RoboDK station: Artist_Larry.rdk

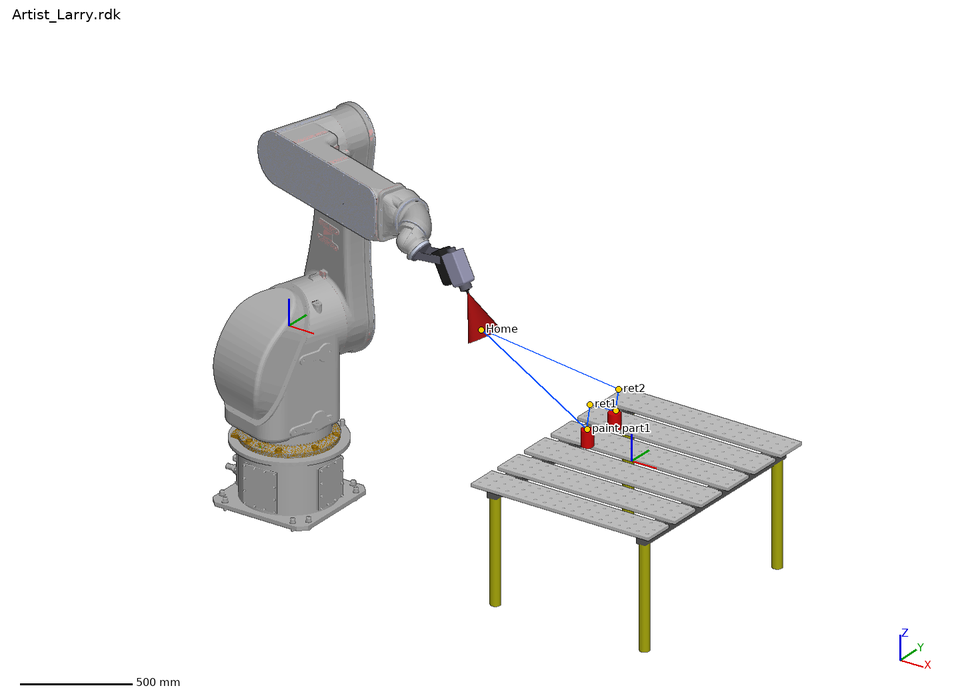
[picture v0: the station drawn from its stored meshes, robots at their saved joint values, targets as dots, program paths as lines]
Station Artist_Larry (saved by RoboDK 5.5.4). Poses are relative to the parent item; angles as X-Y-Z fixed-axis rotations.
Station parameters (name, value as stored): LIN64
  - frame Fanuc P-50iB/10L Base at (0, 0, 0) mm
    - robot Fanuc P-50iB/10L: 6 axes, payload 10 kg, reach 1800 mm, repeatability 0.2 mm, weight 331 kg
        modified DH rows (alpha deg, a mm, theta deg, d mm): 0, 0, 0, 850; -90, 0, -90, 0; 0, 900, 0, 0; -90, 0, -90, 863.603; 70, 0, 0, 106.418; -70, 0, 0, 82
        base shift (0, 0, -850) mm
        joint limits [-160, -45, -205, -360, -360, -360] to [160, 120, 165, 360, 360, 360]; home [0, 0, 0, 0, 0, 0]; saved at [-16.454, 4.54, -1.669, 66.192, 32.539, 108.194]
      - tool Paint gun, TCP at (50, 0, 450) mm, rotated rx 0 ry 30 rz 0 deg, size 203.2 x 279.7 x 471.5 mm
  - frame Frame 2 at (1847.5, 25.56, -163.78) mm
    - object Object Table at (25, 0, 0) mm, rotated rx 0 ry 0 rz 90 deg, size 1193.8 x 965.2 x 609.6 mm, geometry from Object Table.wrl
      - object Part 1 at (-43.87, 237.19, 75.51) mm, size 60 x 60 x 80 mm, geometry from part.sld
      - object Part 2 at (168.08, 237.19, 75.51) mm, size 60 x 60 x 80 mm, geometry from part.sld
    - target Home (Cartesian target) at (-512.99, -434.82, 681.29) mm, rotated rx -177.27 ry 29.43 rz 176.85 deg; joints [-12.777, 34.217, -8.53, 77.216, 55.627, 89.723] of Fanuc P-50iB/10L
    - target paint part1 (Cartesian target) at (-212.06, -43.87, 115.51) mm, rotated rx -180 ry 0 rz 176.85 deg; joints [3.806, 37.835, -17.333, 86.864, 45.873, 71.994] of Fanuc P-50iB/10L
    - target ret1 (Cartesian target) at (-196.3, -42.96, 243.33) mm, rotated rx 179.4 ry 4.87 rz 176.81 deg; joints [3.8, 34.28, -12.43, 86.86, 45.87, 71.99] of Fanuc P-50iB/10L
    - target paint part2 (Cartesian target) at (-215.46, 184.9, 115.51) mm, rotated rx -180 ry 0 rz 176.85 deg; joints [12.99, 38.753, -17.421, 93.025, 47.147, 59.125] of Fanuc P-50iB/10L
    - target ret2 (Cartesian target) at (-201.93, 188.08, 223.02) mm, rotated rx 178.84 ry 3.96 rz 176.8 deg; joints [12.99, 35.77, -13.3, 93.02, 47.14, 59.12] of Fanuc P-50iB/10L
  - program PaintDemo (8 instructions, listed below)
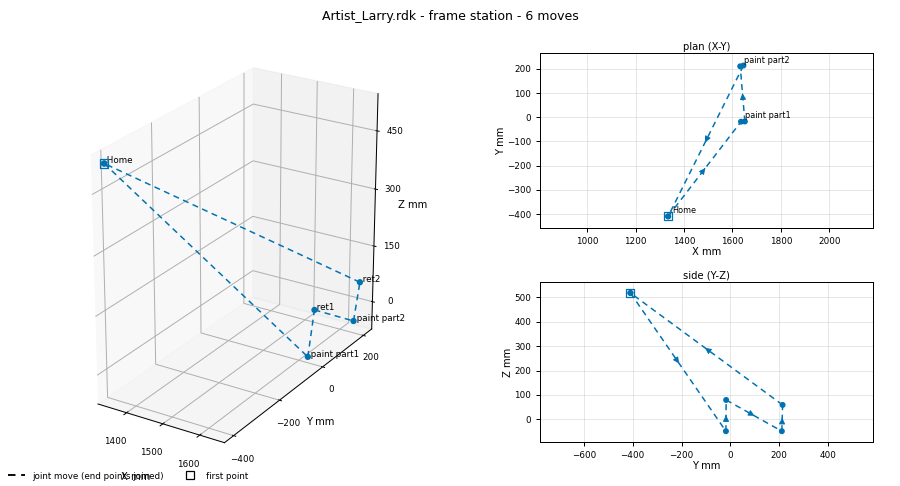
[picture p0: tool path of Artist_Larry.rdk in frame station, 6 of 6 moves have a stored position in this frame; points joined in program order, loops and branches not executed]

--- program PaintDemo (robot Fanuc P-50iB/10L) ---
  Set Ref.: Frame 2
  Set Tool: Paint gun
  MoveJ (Home)
  MoveJ (paint part1)
  MoveJ (ret1)
  MoveJ (paint part2)
  MoveJ (ret2)
  MoveJ (Home)
